FUNCTION_BLOCK ConvertAnyToString_TEST EXTENDS TcUnit.FB_TestSuite
VAR_INPUT
END_VAR
VAR_OUTPUT
END_VAR
VAR
END_VAR

ConvertAnyByteToString();
ConvertAnyDateAndTimeToString();
ConvertAnyDateToString();
ConvertAnyDINTToString();
ConvertAnyDTToString();
ConvertAnyINTToString();
ConvertAnyLINTToString();
ConvertAnyLRealToString();
ConvertAnyLWordToString();
ConvertAnyRealToString();
ConvertAnySINTToString();
ConvertAnyStringToString();
ConvertAnyTimeToString();
ConvertAnyTODToString();
ConvertAnyUDINTToString();
ConvertAnyUINTToString();
ConvertAnyULINTToString();
ConvertAnyUSINTToString();
ConvertAnyWordToString();
ConvertAnyWStringToString();

METHOD _FormatResult : STRING
VAR_INPUT
	expected : STRING; 
	result: STRING;
END_VAR
_FormatResult := CONCAT('Conversion failed. Expected: ', CONCAT(expected, CONCAT(' - Result: ', result)));
END_METHOD

METHOD ConvertAnyByteToString : BOOL
VAR_INPUT
END_VAR
VAR
	input: BYTE := 1;
	result: STRING;
	expected: STRING := '1';
END_VAR
TEST('ConvertAnyByteToString');
 
result := ANY_TO_STRING2(input);
 
AssertEquals(Expected := expected,
             Actual := result,
             Message := _FormatResult(expected, result));
 
TEST_FINISHED();
END_METHOD

METHOD ConvertAnyDateAndTimeToString : BOOL
VAR_INPUT
END_VAR
VAR
	input: DATE_AND_TIME := DT#1970-01-01-00:00;
	result: STRING;
	expected: STRING := 'DT#1970-01-01-00:00:00';
END_VAR
TEST('ConvertAnyDateAndTimeToString');
 
result := ANY_TO_STRING2(input);
 
AssertEquals(Expected := expected,
             Actual := result,
             Message := _FormatResult(expected, result));
 
TEST_FINISHED();
END_METHOD

METHOD ConvertAnyDateToString : BOOL
VAR_INPUT
END_VAR
VAR
	input: DATE := D#1970-01-01;
	result: STRING;
	expected: STRING := 'D#1970-01-01';
END_VAR
TEST('ConvertAnyDateToString');
 
result := ANY_TO_STRING2(input);
 
AssertEquals(Expected := expected,
             Actual := result,
             Message := _FormatResult(expected, result));
 
TEST_FINISHED();
END_METHOD

METHOD ConvertAnyDINTToString : BOOL
VAR_INPUT
END_VAR
VAR
	input: DINT := 1;
	result: STRING;
	expected: STRING := '1';
END_VAR
TEST('ConvertAnyDINTToString');
 
result := ANY_TO_STRING2(input);
 
AssertEquals(Expected := expected,
             Actual := result,
             Message := _FormatResult(expected, result));
 
TEST_FINISHED();
END_METHOD

METHOD ConvertAnyDTToString : BOOL
VAR_INPUT
END_VAR
VAR
	input: DT := DT#1970-01-01-00:00;
	result: STRING;
	expected: STRING := 'DT#1970-01-01-00:00:00';
END_VAR
TEST('ConvertAnyDTToString');
 
result := ANY_TO_STRING2(input);
 
AssertEquals(Expected := expected,
             Actual := result,
             Message := _FormatResult(expected, result));
 
TEST_FINISHED();
END_METHOD

METHOD ConvertAnyDWordToString : BOOL
VAR_INPUT
END_VAR
VAR
	input: DWORD := 1;
	result: STRING;
	expected: STRING := '1';
END_VAR
TEST('ConvertAnyDWordToString');
 
result := ANY_TO_STRING2(input);
 
AssertEquals(Expected := expected,
             Actual := result,
             Message := _FormatResult(expected, result));
 
TEST_FINISHED();
END_METHOD

METHOD ConvertAnyINTToString : BOOL
VAR_INPUT
END_VAR
VAR
	input: INT := 1;
	result: STRING;
	expected: STRING := '1';
END_VAR
TEST('ConvertAnyINTToString');
 
result := ANY_TO_STRING2(input);
 
AssertEquals(Expected := expected,
             Actual := result,
             Message := _FormatResult(expected, result));
 
TEST_FINISHED();
END_METHOD

METHOD ConvertAnyLINTToString : BOOL
VAR_INPUT
END_VAR
VAR
	input: LINT := 1;
	result: STRING;
	expected: STRING := '1';
END_VAR
TEST('ConvertAnyLINTToString');
 
result := ANY_TO_STRING2(input);
 
AssertEquals(Expected := expected,
             Actual := result,
             Message := _FormatResult(expected, result));
 
TEST_FINISHED();
END_METHOD

METHOD ConvertAnyLRealToString : BOOL
VAR_INPUT
END_VAR
VAR
	input: REAL := 1.0;
	result: STRING;
	expected: STRING := '1.0';
END_VAR
TEST('ConvertAnyRealToString');
 
result := ANY_TO_STRING2(input);
 
AssertEquals(Expected := expected,
             Actual := result,
             Message := _FormatResult(expected, result));
 
TEST_FINISHED();
END_METHOD

METHOD ConvertAnyLWordToString : BOOL
VAR_INPUT
END_VAR
VAR
	input: LWORD := 1;
	result: STRING;
	expected: STRING := '1';
END_VAR
TEST('ConvertAnyLWordToString');
 
result := ANY_TO_STRING2(input);
 
AssertEquals(Expected := expected,
             Actual := result,
             Message := _FormatResult(expected, result));
 
TEST_FINISHED();
END_METHOD

METHOD ConvertAnyRealToString : BOOL
VAR_INPUT
END_VAR
VAR
	input: LREAL := 1.0;
	result: STRING;
	expected: STRING := '1.0';
END_VAR
TEST('ConvertAnyLRealToString');
 
result := ANY_TO_STRING2(input);
 
AssertEquals(Expected := expected,
             Actual := result,
             Message := _FormatResult(expected, result));
 
TEST_FINISHED();
END_METHOD

METHOD ConvertAnySINTToString : BOOL
VAR_INPUT
END_VAR
VAR
	input: SINT := 1;
	result: STRING;
	expected: STRING := '1';
END_VAR
TEST('ConvertAnySINTToString');
 
result := ANY_TO_STRING2(input);
 
AssertEquals(Expected := expected,
             Actual := result,
             Message := _FormatResult(expected, result));
 
TEST_FINISHED();
END_METHOD

METHOD ConvertAnyStringToString : BOOL
VAR_INPUT
END_VAR
VAR
	input: STRING := 'Hallo';
	result: STRING;
	expected: STRING := 'Hallo';
END_VAR
TEST('ConvertAnyStringToString');
 
result := ANY_TO_STRING2(input);
 
AssertEquals(Expected := expected,
             Actual := result,
             Message := _FormatResult(expected, result));
 
TEST_FINISHED();
END_METHOD

METHOD ConvertAnyTimeToString : BOOL
VAR_INPUT
END_VAR
VAR
	input: TIME := T#49D17H2M47S295MS;
	result: STRING;
	expected: STRING := 'T#49d17h2m47s295ms';
END_VAR
TEST('ConvertAnyTimeToString');
 
result := ANY_TO_STRING2(input);
 
AssertEquals(Expected := expected,
             Actual := result,
             Message := _FormatResult(expected, result));
 
TEST_FINISHED();
END_METHOD

METHOD ConvertAnyTODToString : BOOL
VAR_INPUT
END_VAR
VAR
	input: TOD := TOD#11:02:47.295;
	result: STRING;
	expected: STRING := 'TOD#11:02:47.295';
END_VAR
TEST('ConvertAnyTODToString');
 
result := ANY_TO_STRING2(input);
 
AssertEquals(Expected := expected,
             Actual := result,
             Message := _FormatResult(expected, result));
 
TEST_FINISHED();
END_METHOD

METHOD ConvertAnyUDINTToString : BOOL
VAR_INPUT
END_VAR
VAR
	input: UDINT := 1;
	result: STRING;
	expected: STRING := '1';
END_VAR
TEST('ConvertAnyUDINTToString');
 
result := ANY_TO_STRING2(input);
 
AssertEquals(Expected := expected,
             Actual := result,
             Message := _FormatResult(expected, result));
 
TEST_FINISHED();
END_METHOD

METHOD ConvertAnyUINTToString : BOOL
VAR_INPUT
END_VAR
VAR
	input: UINT := 1;
	result: STRING;
	expected: STRING := '1';
END_VAR
TEST('ConvertAnyUINTToString');
 
result := ANY_TO_STRING2(input);
 
AssertEquals(Expected := expected,
             Actual := result,
             Message := _FormatResult(expected, result));
 
TEST_FINISHED();
END_METHOD

METHOD ConvertAnyULINTToString : BOOL
VAR_INPUT
END_VAR
VAR
	input: ULINT := 1;
	result: STRING;
	expected: STRING := '1';
END_VAR
TEST('ConvertAnyULINTToString');
 
result := ANY_TO_STRING2(input);
 
AssertEquals(Expected := expected,
             Actual := result,
             Message := _FormatResult(expected, result));
 
TEST_FINISHED();
END_METHOD

METHOD ConvertAnyUSINTToString : BOOL
VAR_INPUT
END_VAR
VAR
	input: USINT := 1;
	result: STRING;
	expected: STRING := '1';
END_VAR
TEST('ConvertAnyUSINTToString');
 
result := ANY_TO_STRING2(input);
 
AssertEquals(Expected := expected,
             Actual := result,
             Message := _FormatResult(expected, result));
 
TEST_FINISHED();
END_METHOD

METHOD ConvertAnyWordToString : BOOL
VAR_INPUT
END_VAR
VAR
	input: WORD := 1;
	result: STRING;
	expected: STRING := '1';
END_VAR
TEST('ConvertAnyWordToString');
 
result := ANY_TO_STRING2(input);
 
AssertEquals(Expected := expected,
             Actual := result,
             Message := _FormatResult(expected, result));
 
TEST_FINISHED();
END_METHOD

METHOD ConvertAnyWStringToString : BOOL
VAR_INPUT
END_VAR
VAR
	input: WSTRING := "Hallo";
	result: STRING;
	expected: STRING := 'Hallo';
END_VAR
TEST('ConvertAnyWStringToString');
 
result := ANY_TO_STRING2(input);
 
AssertEquals(Expected := expected,
             Actual := result,
             Message := _FormatResult(expected, result));
 
TEST_FINISHED();
END_METHOD

END_FUNCTION_BLOCK

(* stored: Version 1.1.0.1
   POU ConvertAnyToString_TEST: Id {c0c8c635-4bd3-4a6c-aa53-91d1d9ba5250}, SpecialFunc None
   Method _FormatResult: Id {ac709183-84fd-46b2-8c6b-eae248cb6f14}
   Method ConvertAnyByteToString: Id {eb3ebb05-ad14-4014-b181-b83ce5dcc375}
   Method ConvertAnyDateAndTimeToString: Id {3ceb2e55-4c60-46bd-b69f-89df47ade6d1}
   Method ConvertAnyDateToString: Id {ac53b27f-19f0-4597-a6b1-0978a63259bd}
   Method ConvertAnyDINTToString: Id {41f0e337-a99d-4a1d-a418-57f59f884535}
   Method ConvertAnyDTToString: Id {fff84db2-9556-4bcf-a7c2-65175a561709}
   Method ConvertAnyDWordToString: Id {7a44293c-9be6-4708-958d-b8ccd6433e03}
   Method ConvertAnyINTToString: Id {d3445b3a-c4f0-496c-8c84-057baa011718}
   Method ConvertAnyLINTToString: Id {dc286609-7e6a-4833-a6e2-95f800a2af48}
   Method ConvertAnyLRealToString: Id {92605265-e930-4f9a-99dd-3badfd92d652}
   Method ConvertAnyLWordToString: Id {98dd4e4c-d15f-4397-8faf-efbb8dfd20bb}
   Method ConvertAnyRealToString: Id {c2a19236-c97e-4f2e-a561-eb788168efbf}
   Method ConvertAnySINTToString: Id {6c66c3fb-11c9-4519-ae5e-0bb7f858bd6f}
   Method ConvertAnyStringToString: Id {4c0e1966-ea45-465b-b9de-b0deb0eb467f}
   Method ConvertAnyTimeToString: Id {e48b511f-76fd-4678-bbd2-4c20b28dd6bb}
   Method ConvertAnyTODToString: Id {69944400-4089-476f-a2de-3ad376c4053f}
   Method ConvertAnyUDINTToString: Id {91b5769e-d98f-4867-9e1e-6d987069ea4a}
   Method ConvertAnyUINTToString: Id {8ae38335-329f-4d9c-ab53-af988e6cceac}
   Method ConvertAnyULINTToString: Id {eb9b2ce1-3cd2-4ea0-89a9-45bc991095e1}
   Method ConvertAnyUSINTToString: Id {12bcc65b-08b3-4fa4-9ece-e0c6dfb096e6}
   Method ConvertAnyWordToString: Id {ef1c000d-a9e4-4adc-bf4d-87ef6c426de0}
   Method ConvertAnyWStringToString: Id {914107a8-aa4b-4098-9f38-02385e7c4de4} *)
